# EPICS StreamDevice protocol: CavitySimulator-loc/CavitySimulatorApp/Db/EEPROM.proto
# EEPROM protocols

ExtraInput = Ignore;
InTerminator = NL;
OutTerminator = NL"*OPC?"NL;

save { out "SET:SAVE";}

get { out "SET:RESTORE";}
